TYPE TestReportHandle_t : Pointer to FB_TestReportBase; END_TYPE

(* stored: Version 1.1.0.1, ProductVersion 3.1.4024.12
   DUT TestReportHandle_t: Id {7106b689-a75c-400e-a8fa-9e258dd8cf30} *)
